FUNCTION_BLOCK FB_HMIManager EXTENDS FB_BaseGroupElement IMPLEMENTS ITF_HMIManager
VAR
END_VAR

END_FUNCTION_BLOCK

(* stored: Version 1.1.0.1
   POU FB_HMIManager: Id {a88b626b-1335-01ba-387a-b90d8f220c55}, SpecialFunc None *)
